INTERFACE IPid

PROPERTY DifferentialPartLimit : LREAL
SET
END_SET
END_PROPERTY

PROPERTY PreviousIntegralPart : LREAL
SET
END_SET
END_PROPERTY

END_INTERFACE

(* stored: Version 1.1.0.1, ProductVersion 3.1.4024.12
   Itf IPid: Id {8da9abfe-226e-4374-8b8c-042275335040}
   Property DifferentialPartLimit: Id {6b409b6c-e5da-47f3-8c78-be6455f35001}
   Set Set: Id {fb1af68a-7410-4ee6-a26f-da9cb38e3c8d}
   Property PreviousIntegralPart: Id {a71b62c7-c254-4773-b8fa-48b59422a176}
   Set Set: Id {ac35ef80-707b-4fe3-b090-b8f4674b975e} *)
